Fanuc KAREL source: ka00012.KL

PROGRAM KA00012
%NOLOCKGROUP
VAR
SRC:INTEGER
DST : ARRAY[2] OF SHORT
BEGIN
SRC=2
DST[1]=SRC
END KA00012
